INTERFACE ITF_BaseComponent_HMI EXTENDS ITF_BaseLoggerElement_HMI

METHOD PUBLIC IsValidCommonData : BOOL
VAR_INPUT
END_VAR
END_METHOD

METHOD PUBLIC LinkCommonData : BOOL
VAR_INPUT
	stCommonData				: REFERENCE TO ST_BaseCommonData;
END_VAR
END_METHOD

END_INTERFACE

(* stored: Version 1.1.0.1
   Itf ITF_BaseComponent_HMI: Id {09893359-9aae-0055-210b-9fb2bfb82b06}
   Method IsValidCommonData: Id {3f7a8c5a-8eb8-0328-2fa4-dbdaa99c550b}
   Method LinkCommonData: Id {9592f34a-d939-01f0-03b2-89c41fa48d7d} *)
